{attribute 'linkalways'} 
{attribute 'no_explicit_call' := 'This FB is a CLASS and must be accessed using methods or properties'}
{attribute 'enable_dynamic_creation'}
FUNCTION_BLOCK Node_ContainerType_Vector_TcVnVector4_SINT EXTENDS Node
VAR
    out : _GUID;
END_VAR

METHOD PUBLIC  Clone : I_Node
VAR
	pNode : POINTER TO Node_ContainerType_Vector_TcVnVector4_SINT;
END_VAR
pNode := __NEW(Node_ContainerType_Vector_TcVnVector4_SINT);
Clone := pNode^;
END_METHOD

METHOD FB_init : BOOL
VAR_INPUT
	bInitRetains : BOOL; // if TRUE, the retain variables are initialized (warm start / cold start)
	bInCopyCode : BOOL;  // if TRUE, the instance afterwards gets moved into the copy code (online change)
END_VAR
AddOutput('out', out);
END_METHOD

METHOD PROTECTED OnExecute
out.Value := ContainerType_Vector_TcVnVector4_SINT;
END_METHOD

END_FUNCTION_BLOCK

(* stored: Version 1.1.0.1, ProductVersion 3.1.4026.17
   POU Node_ContainerType_Vector_TcVnVector4_SINT: Id {6f05e4a6-b3c8-050a-1866-e6c03b05ddbf}, SpecialFunc None
   Folder Constructor: Id {c9d54440-c753-0012-0530-7f3c84cb14f7}
   Method Clone: Id {61da00cb-4028-05d8-2a34-76bef98c031d}
   Method FB_init: Id {642fea00-9ba7-049e-2fca-dbb20b30fbda}
   Method OnExecute: Id {051d70aa-415e-0ae2-2972-a02050bdbcd7} *)
